// TIA Portal V17 export
// export: Created 2025-03-10T12:15:07.0536311Z, ExportSetting WithDefaults, DisplayName Totally Integrated Automation Portal, DisplayVersion V17 Update 8, DisplayName TIA Portal Openness, DisplayVersion V17 Update 8, DisplayName TIA Portal Version Control Interface, DisplayVersion V17, DisplayName SINAMICS Startdrive Advanced, DisplayVersion V17 SP2, DisplayName SINAMICS Startdrive G110M, G120, G120C, G120D, G120P, G115D, DisplayVersion V17 SP2, DisplayName SINAMICS Startdrive G130, G150, S120, S150, SINAMICS MV, S210, DisplayVersion V17 SP2, DisplayName STEP 7 Professional, DisplayVersion V17 Update 8, DisplayName SINUMERIK ONE STEP 7 Toolbox, DisplayVersion V17 Update 12, DisplayName SINUMERIK 840D sl STEP 7 Toolbox, DisplayVersion V17 Update 12, DisplayName STEP 7 Safety, DisplayVersion V17 Update 6, DisplayName WinCC Advanced, DisplayVersion V17 Update 8
DATA_BLOCK "DB7400_QUALITY"   // DB7400
{ S7_Optimized_Access := 'FALSE'; DB_Accessible_From_OPC_UA := 'FALSE' }
AUTHOR : ETXETAR
VERSION : 1.0
// stored: AutoNumber false, DBAccessibleFromOPCUA false, DBAccessibleFromWebserver true, IsOnlyStoredInLoadMemory false, IsWriteProtectedInAS false
   VAR RETAIN
      OPTIONS : Struct   // OPTIONS
         QC_STOP_END_OF_CYCLE : Bool;   // QC STOP END OF CYCLE
         SP11_WORKS_TWO_PARTS : Bool;   // SP11 WORKS TWO PARTS
         SP12_WORKS_TWO_PARTS : Bool;   // SP12 WORKS TWO PARTS
         SP21_WORKS_TWO_PARTS : Bool;   // SP21 WORKS TWO PARTS
         SP22_WORKS_TWO_PARTS : Bool;   // SP22 WORKS TWO PARTS
         FIRST_SCAN : Bool;   // FIRST SCAN
         CYCLE_INTERRUPTED : Bool;   // CYCLE INTERRUPTED
         ANY_TOOL_NEW : Bool;   // ANY TOOL NEW
         BROKEN_TOOL : Bool;   // BROKEN TOOL
         ALL_BROKEN_TOOL : Bool;   // ALL BROKEN TOOL IF ONE TOOL IS BROKEN ALL PARTS ARE MARKED
         ONE_COUNTER : Bool;   // ONE COUNTER
         COUNTER_PER_PART : Bool;   // COUNTER PER PART
         CMM_QUALITY_CHECK : Bool;   // CMM QUALITY CHECK
         SURFACE_QUALITY_CHECK : Bool;   // SURFACE QUALITY CHECK
      END_STRUCT;
      PART_CONTROL : Struct   // PART CONTROL
         HMI_QUALITY_HALF_PART : Bool;   // HMI QUALITY HALF PART
         HMI_QUALITY_FULL_PART : Bool;   // HMI QUALITY FULL PART
         HMI_QUALITY_CANCEL : Bool;   // HMI QUALITY CANCEL
         HMI_QUALITY_NOK : Bool;   // HMI QUALITY NOK
         HMI_QUALITY_OK : Bool;   // HMI QUALITY OK
         HALF_QUALITY_PART_SELECTED : Bool;   // HALF QUALITY PART SELECTED
         FULL_QUALITY_PART_SELECTED : Bool;   // FULL QUALITY PART SELECTED
         PART_QUALITY_ON_DEMAND : Bool;   // PART QUALITY ON DEMAND
         QUALITY_AUX_WARNING : Bool;   // QUALITY AUX WARNING
         QUALITY_AUX_FAULT : Bool;   // QUALITY AUX FAULT
         QUALITY_PART : Bool;   // QUALITY PART
         FIXTURE_2_QUALITY : Bool;   // FIXTURE 2 QUALITY
         U01_FIXTURE_1_PART_P : Bool;   // UNIT 01 FIXTURE 1 PART A PULSE
         U01_FIXTURE_2_PART_P : Bool;   // UNIT 01 FIXTURE 2 PART A PULSE
         U01_FIXTURE_3_PART_P : Bool;   // UNIT 01 FIXTURE 3 PART A PULSE
         U01_FIXTURE_4_PART_P : Bool;   // UNIT 01 FIXTURE 4 PART A PULSE
         U02_FIXTURE_1_PART_P : Bool;   // UNIT 02 FIXTURE 1 PART A PULSE
         U02_FIXTURE_2_PART_P : Bool;   // UNIT 02 FIXTURE 2 PART A PULSE
         U02_FIXTURE_3_PART_P : Bool;   // UNIT 02 FIXTURE 3 PART A PULSE
         U02_FIXTURE_4_PART_P : Bool;   // UNIT 02 FIXTURE 4 PART A PULSE
         U01_FIXTURE_1_PART_DEMAND : Bool;   // UNIT 01 FIXTURE 1 PART A DEMAND
         U01_FIXTURE_2_PART_DEMAND : Bool;   // UNIT 01 FIXTURE 2 PART A DEMAND
         U01_FIXTURE_3_PART_DEMAND : Bool;   // UNIT 01 FIXTURE 3 PART A DEMAND
         U01_FIXTURE_4_PART_DEMAND : Bool;   // UNIT 01 FIXTURE 4 PART A DEMAND
         U02_FIXTURE_1_PART_DEMAND : Bool;   // UNIT 02 FIXTURE 1 PART A DEMAND
         U02_FIXTURE_2_PART_DEMAND : Bool;   // UNIT 02 FIXTURE 2 PART A DEMAND
         U02_FIXTURE_3_PART_DEMAND : Bool;   // UNIT 02 FIXTURE 3 PART A DEMAND
         U02_FIXTURE_4_PART_DEMAND : Bool;   // UNIT 02 FIXTURE 4 PART A DEMAND
         PART_NOK : Bool;   // PART QUALITY DEMAND NOK ALARM
      END_STRUCT;
      PART_TYPE : Struct   // PART TYPE
         PART_TYPE_CHANGE_AUX : Bool;   // PART TYPE CHANGE AUXILIARY
         FIXTURE_1_PART_TYPE_CHANGE : Bool;   // FIXTURE 1 PART TYPE CHANGE
         FIXTURE_2_PART_TYPE_CHANGE : Bool;   // FIXTURE 2 PART TYPE CHANGE
         FIXTURE_3_PART_TYPE_CHANGE : Bool;   // FIXTURE 3 PART TYPE CHANGE
         FIXTURE_4_PART_TYPE_CHANGE : Bool;   // FIXTURE 4 PART TYPE CHANGE
         QUALITY_PART_TYPE_CHANGE : Bool;   // QUALITY AFTER PART TYPE CHANGE
         QUALITY_PART_NOK : Bool;   // QUALITY PART AFTER PART TYPE CHANGE NOK ALARM
      END_STRUCT;
      FIRST_CYCLE : Struct   // FIRST CYCLE
         FIRST_SCAN_AUX : Bool;   // FIRST SCAN AUXILIARY
         QUALITY_FIRST_CYCLE : Bool;   // QUALITY FIRST CYCLE
         FIXTURE_2_FIRST_CYCLE : Bool;   // FIXTURE 2 FIRST CYCLE
         FIXTURE_1_PART_A : Bool;   // FIXTURE 1 PART A FIRST CYCLE
         FIXTURE_1_PART_A_NOK : Bool;   // FIXTURE 1 PART A FIRST CYCLE NOK ALARM
      END_STRUCT;
      CYCLE_INTERRUPTED : Struct   // CYCLE INTERRUPTED
         CYCLE_INTERRUPTED_AUX : Bool;   // CYCLE INTERRUPTED AUXILIARY
         CYCLE_INTERRUPTED_AUX_P : Bool;   // CYCLE INTERRUPTED AUXILIARY PULSE
         FIXTURE_1_CYCLE_INTERRUPTED : Bool;   // FIXTURE 1 CYCLE INTERRUPTED
         FIXTURE_2_CYCLE_INTERRUPTED : Bool;   // FIXTURE 2 CYCLE INTERRUPTED
         FIXTURE_1_PART_A : Bool;   // FIXTURE 1 PART A CYCLE INTERRUPTED
         FIXTURE_1_PART_B : Bool;   // FIXTURE 1 PART B CYCLE INTERRUPTED
         FIXTURE_1_PART_C : Bool;   // FIXTURE 1 PART C CYCLE INTERRUPTED
         FIXTURE_1_PART_D : Bool;   // FIXTURE 1 PART D CYCLE INTERRUPTED
         FIXTURE_2_PART_A : Bool;   // FIXTURE 2 PART A CYCLE INTERRUPTED
         FIXTURE_2_PART_B : Bool;   // FIXTURE 2 PART B CYCLE INTERRUPTED
         FIXTURE_2_PART_C : Bool;   // FIXTURE 2 PART C CYCLE INTERRUPTED
         FIXTURE_2_PART_D : Bool;   // FIXTURE 2 PART D CYCLE INTERRUPTED
         FIXTURE_1_PART_A_NOK : Bool;   // FIXTURE 1 PART A CYCLE INTERRUPTED NOK ALARM
         FIXTURE_1_PART_B_NOK : Bool;   // FIXTURE 1 PART B CYCLE INTERRUPTED NOK ALARM
         FIXTURE_1_PART_C_NOK : Bool;   // FIXTURE 1 PART C CYCLE INTERRUPTED NOK ALARM
         FIXTURE_1_PART_D_NOK : Bool;   // FIXTURE 1 PART D CYCLE INTERRUPTED NOK ALARM
         FIXTURE_2_PART_A_NOK : Bool;   // FIXTURE 2 PART A CYCLE INTERRUPTED NOK ALARM
         FIXTURE_2_PART_B_NOK : Bool;   // FIXTURE 2 PART B CYCLE INTERRUPTED NOK ALARM
         FIXTURE_2_PART_C_NOK : Bool;   // FIXTURE 2 PART C CYCLE INTERRUPTED NOK ALARM
         FIXTURE_2_PART_D_NOK : Bool;   // FIXTURE 2 PART D CYCLE INTERRUPTED NOK ALARM
         S_PECT_01 : TP_TIME;   // S PECT 01
      END_STRUCT;
      PART_COUNTER : Struct   // PART COUNTER
         PART_COUNTER_REACHED_AUX : Bool;   // PART COUNTR REACHED AUXILIARY
         PARTS_COUNTER_AUX_P : Bool;   // PARTS COUNTER AUX PULSE
         QUALITY_PART_COUNTER_REACHED : Bool;   // QUALITY AFTER PART COUNTER REACHED
         QUALITY_PART_NOK : Bool;   // QUALITY PART AFTER PART COUNTER REACHED ALARM
      END_STRUCT;
      QUALITY_AUX_DATA : Struct   // QUALITY AUXILIARY DATA
         PARTS_COUNTER : Int := 0;   // PARTS COUNTER
         QUALITY_AFTER_PARTS : Int;   // PARTS BEFORE CHECK QUALITY
      END_STRUCT;
   END_VAR
BEGIN
END_DATA_BLOCK
